TYPE CmpConvMergeConfig :
STRUCT
	BufferSensorOnTime: TIME;
	BufferSensorOffTime: TIME;
	MergeTimeSpacing: TIME;
	MergeTimeMainTravel: TIME;
	MergeTimeSpurTravel: TIME;
	UseReleaseRatio: BOOL;
	RatioMain: REAL;
	RatioSpur: REAL;
END_STRUCT
END_TYPE

(* stored: Version 1.1.0.1, ProductVersion 3.1.4024.6
   DUT CmpConvMergeConfig: Id {3e122273-ff54-4dd9-a87b-3d02017189ac} *)
